// TIA Portal V20 export
DATA_BLOCK "T1-A ARUNC"   // DB1102
{ S7_Optimized_Access := 'TRUE' }
AUTHOR : SAS
// stored: AutoNumber false, IsRetainMemResEnabled true, MemoryReserve 100, RetainMemoryReserve 100
   VAR RETAIN
      "Seq Status" : Struct
         ReadyToAuto : Bool;
         AutoON : Bool;
         WaitPiece : Bool;
         Stopped : Bool;
         "Step" : Struct
            Actual : Int;
            "-1" : Int;
            "-2" : Int;
            "-3" : Int;
            "-4" : Int;
            "-5" : Int;
            "-6" : Int;
            "-7" : Int;
            "-8" : Int;
            "-9" : Int;
            "Actual time" : Time_Of_Day;
            "-1 Time" : Time_Of_Day;
            "-2 Time" : Time_Of_Day;
            "-3 Time" : Time_Of_Day;
            "-4 Time" : Time_Of_Day;
            "-5 Time" : Time_Of_Day;
            "-6 Time" : Time_Of_Day;
            "-7 Time" : Time_Of_Day;
            "-8 Time" : Time_Of_Day;
            "-9 Time" : Time_Of_Day;
         END_STRUCT;
      END_STRUCT;
      Transitions : Struct
         Safe : Bool;   // Emergency
         Fault : Bool;   // Fault
         Auto : Bool;
         Manual : Bool;
         Pause : Bool;
         Stop : Bool;
         "Cycle start request" : Bool;
         "First Piece" : Bool;
         "Piece presence" : Bool;
         "Adjacent Machines" : Bool;
         "Adjacent Machines Repositioning" : Bool;   // Only for repositioning
         Init_Sequence : Bool;
         "Movement conditions 1" : Bool;   // Load
         "Movement conditions 2" : Bool;
         "Movement conditions 3" : Bool;
         "Movement conditions 4" : Bool;
         "Reset Fault" : Bool;
         "Bypass ilock" : Bool;
      END_STRUCT;
      Memory : Struct
         "Piece presence" : Bool;   // Cumulative piece presence
         "Piece absence" : Bool;   // No sensor triggered
         p2 : Bool;
         "Pipe Transfered" : Bool;   // Pipe transfered
         p4 : Bool;
         "Permanent Condition" : Bool;   // Permanent condition
         "Movement Fault" : Bool;   // Cumulative of Machine Fault condition
         "Local StopAuto" : Bool;   // Local StopAuto
         "Interlocks UP" : Bool;   // Interlocks for UP
         "Interlocks DOWN" : Bool;   // Interlocks for DOWN
         I2 : Bool;
         I3 : Bool;
         I4 : Bool;
         I5 : Bool;
         Mode_change_ready : Bool;   // Machine ready to cheange operation mode (Enable, Disable, LEV2 Auto)
         m1 : Bool;
         m2 : Bool;
         m3 : Bool;
         FW_ON : Bool;   // Flipper RUN
         "Position UP" : Bool;   // Position UP
         "Position DOWN" : Bool;   // Position DOWN
         "Command Scuturator" : Bool;   // Scuturator Comanda
         r0 : Real;
         r1 : Real;
         r2 : Real;
         r3 : Real;
         r4 : Real;
         r5 : Real;
      END_STRUCT;
   END_VAR
BEGIN
END_DATA_BLOCK
